FUNCTION F_TimeStamp13_TO_SYSTEMTIME : TimeStruct
VAR_INPUT
	iUnixTimeStamp13 : ULINT;
END_VAR
VAR
	_FileTime64 :T_FILETIME64;
END_VAR

_FileTime64 := (iUnixTimeStamp13 + 11644473600000 - 5000) * 10000;
F_TimeStamp13_TO_SYSTEMTIME := FILETIME64_TO_SYSTEMTIME(_FileTime64);

END_FUNCTION

(* stored: Version 1.1.0.1, ProductVersion 3.1.4024.12
   POU F_TimeStamp13_TO_SYSTEMTIME: Id {cf181f6a-4a9c-464c-b58a-d3129f2009da}, SpecialFunc None *)
